SUBAPPLICATION Softkey_T_FF_ILOCK_TO_QX_BG (* Digitaler Ausgang als Softkey-Toggle-Flip-Flop (Taste kippt QX) mit zusaetzlichem externen SET/RESET zur Verriegelung, Background spiegelt den Zustand. Generisch. *)
  (* Standard: 61499-2 *)
  (* Version 1.0, 2026-09-09, Franz Höpfinger, Meisterschulen am Ostbahnhof, Ausgelagert aus Uebung_039a_sub_Outputs zur Wiederverwendung. *)
  PACKAGE MyLib::sys;
  IMPORT isobus::UT::io::Softkey::SoftKeyActivationCode::SK_RELEASED;
  IMPORT isobus::UT::Q::const::IDs::ID_NULL;
  IMPORT logiBUS::io::DQ::logiBUS_DO;
  IMPORT logiBUS::io::DQ::logiBUS_DO_S;
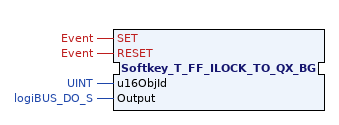
  EVENT_INPUT
    SET; (* Set Output *)
    RESET; (* Reset Output *)
  END_EVENT
  VAR_INPUT
    u16ObjId : UINT := ID_NULL; (* Object ID Softkey/Button *)
    Output : logiBUS::io::DQ::logiBUS_DO_S := logiBUS_DO::Invalid;
  END_VAR
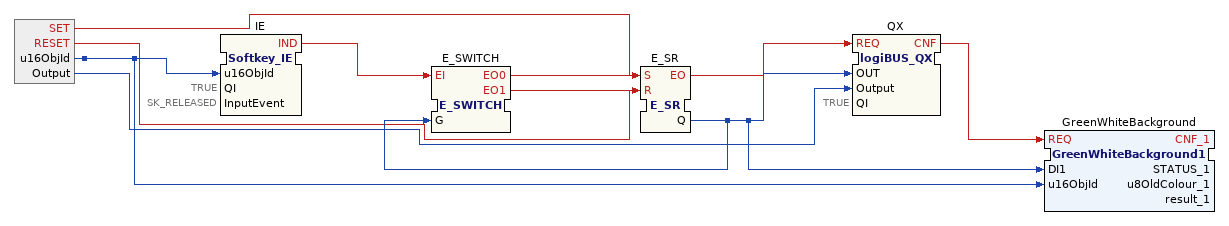
  FBS
    QX : logiBUS::io::DQ::logiBUS_QX(QI := TRUE);
    E_SWITCH : iec61499::events::E_SWITCH;
    E_SR : iec61499::events::E_SR;
    IE : isobus::UT::io::Softkey::Softkey_IE(QI := TRUE, InputEvent := SK_RELEASED);
  END_FBS
  SUBAPPS
    GreenWhiteBackground : MyLib::sys::GreenWhiteBackground1;
  END_SUBAPPS
  EVENT_CONNECTIONS
    QX.CNF TO GreenWhiteBackground.REQ;
    E_SWITCH.EO0 TO E_SR.S;
    E_SWITCH.EO1 TO E_SR.R;
    IE.IND TO E_SWITCH.EI;
    E_SR.EO TO QX.REQ;
    SET TO E_SR.S;
    RESET TO E_SR.R;
  END_CONNECTIONS
  DATA_CONNECTIONS
    u16ObjId TO GreenWhiteBackground.u16ObjId;
    E_SR.Q TO E_SWITCH.G;
    E_SR.Q TO QX.OUT;
    E_SR.Q TO GreenWhiteBackground.DI1;
    u16ObjId TO IE.u16ObjId;
    Output TO QX.Output;
  END_CONNECTIONS
END_SUBAPPLICATION
